{attribute 'qualified_only'}
VAR_GLOBAL
	// Encoder reference values in counts = nm
	nYUP_ENC_REF : ULINT := 14897597;
	nYDWN_ENC_REF : ULINT := 14551600;
	nXUP_ENC_REF : ULINT := 23972500;
	nXDWN_ENC_REF : ULINT := 24766500;
END_VAR

(* stored: Version 1.1.0.1, ProductVersion 3.1.4022.12
   GVL GVL_M2L0: Id {4a614dee-abd1-444d-a31b-b784e14a5b68} *)
